FUNCTION_BLOCK FB_Module01 EXTENDS FB_Module
VAR_INPUT
END_VAR
VAR_OUTPUT
END_VAR
VAR
END_VAR

// https://peterzerlauth.com/
SUPER^();

METHOD PROTECTED M_Execute : BOOL
VAR_INPUT
END_VAR
VAR
	bReturn:					BOOL:= TRUE;
END_VAR
M_Execute:= TRUE;
END_METHOD

METHOD PROTECTED M_Running
VAR_INPUT
END_VAR
END_METHOD

METHOD PROTECTED M_Starting : BOOL
VAR_INPUT
END_VAR
M_Starting:= SUPER^.M_Starting();
END_METHOD

METHOD PROTECTED M_Stopping : BOOL // Return state complete
VAR_INPUT
END_VAR
// State Stopping
M_Stopping:= SUPER^.M_Stopping();
END_METHOD

END_FUNCTION_BLOCK

(* stored: Version 1.1.0.1
   POU FB_Module01: Id {3744d03d-359c-4ab8-84fb-4ea93b7a5162}, SpecialFunc None
   Method M_Execute: Id {0f7f4331-8af5-0744-015a-f65d0021dd06}
   Method M_Running: Id {eaffebca-5ff2-4f17-be84-3310a9ace22e}
   Method M_Starting: Id {6f002794-61fc-043c-1d84-a8bc502c5d3a}
   Method M_Stopping: Id {478c517c-d184-0eaf-2697-597088f6cf3f} *)
